// TIA Portal V18 export
DATA_BLOCK "PLCtoMES"   // DB500
{ S7_Optimized_Access := 'FALSE' }
// stored: AutoNumber false
   VAR
      "PLC.Load_Station1ChickInReq" : Bool;   // 本站工位1打标工位主零件RFID码读出，请求查询
      "PLC.Load_Station2ChickInReq" : Bool;   // 本站工位2贴标工位主零件RFID码读出，请求查询
      "PLC.Load_Station3ChickInReq" : Bool;   // Spare
      "PLC.Load_Station4ChickInReq" : Bool;   // Spare
      "PLC.Load_Station5ChickInReq" : Bool;   // Spare
      "PLC.Load_Station6ChickInReq" : Bool;   // Spare
      "PLC.Load_Station7ChickInReq" : Bool;   // Spare
      "PLC.Load_Station8ChickInReq" : Bool;   // Spare
      "PLC.Load_StoveCheckIn" : Bool;   // 子零件1码读出，请求查询
      Spare_11 : Bool;   // Spare
      Spare_12 : Bool;   // Spare
      Spare_13 : Bool;   // Spare
      Spare_14 : Bool;   // Spare
      Spare_15 : Bool;   // Spare
      Spare_16 : Bool;   // Spare
      Spare_17 : Bool;   // Spare
      Spare_18 : Bool;   // 手持扫码枪1上料查询触发
      Spare_19 : Bool;   // Spare
      Spare_20 : Bool;   // Spare
      Spare_21 : Bool;   // Spare
      Spare_22 : Bool;   // Spare
      Spare_23 : Bool;   // Spare
      Spare_24 : Bool;   // Spare
      Spare_25 : Bool;   // Spare
      Spare_1 : Byte;   // Spare
      Spare_2 : Bool;   // 请求下发打标数据触发
      Spare_3 : Bool;   // 二维码内容与主零件码比对请求
      Spare_4 : Bool;   // Spare
      Spare_5 : Bool;   // Spare
      Spare_6 : Bool;   // Spare
      Spare_7 : Bool;   // Spare
      Spare_8 : Bool;   // Spare
      Spare_9 : Bool;   // Spare
      Spare_10 : Bool;
      Static_2 : Bool;   // 本站工位1打标过程数据保存触发位
      "PLC.Unload_Station1DataSaveReq" : Bool;   // 本站工位2贴标过程数据保存触发位
      "PLC.Unload_Station2DataSaveReq" : Bool;   // Spare
      "PLC.Unload_Station3DataSaveReq" : Bool;   // Spare
      "PLC.Unload_Station4DataSaveReq" : Bool;   // Spare
      "PLC.Unload_Station5DataSaveReq" : Bool;   // Spare
      "PLC.Unload_Station6DataSaveReq" : Bool;   // Spare
      "PLC.Unload_Station7DataSaveReq" : Bool;   // Spare
      "PLC.Unload_Station8DataSaveReq" : Bool;   // PLC心跳
      "PLC.Unload_HeartbeatSignal" : Bool;
   END_VAR
BEGIN
END_DATA_BLOCK
